(* IEC 61131-3 sources: stc/tests/fixtures/valid_codegen, 3 files *)

(* ---- not_equal.st ---- *)
(* Copyright (C) 2021-2026 Manuele Conti
   SPDX-License-Identifier: GPL-2.0-or-later
   Summary: Verifies code generation for the IEC not-equal operator. *)

FUNCTION differs : BOOL
VAR_INPUT
    left_value, right_value: INT;
END_VAR
    differs := left_value <> right_value;
END_FUNCTION

(* ---- repeat_loop.st ---- *)
(* Copyright (C) 2021-2026 Manuele Conti
   SPDX-License-Identifier: GPL-2.0-or-later
   Summary: Verifies code generation for REPEAT iteration. *)

FUNCTION climb_until : INT
VAR_INPUT
    start_value: INT;
END_VAR
VAR
    cursor_value: INT;
END_VAR
    cursor_value := start_value;
    REPEAT
        cursor_value := cursor_value + 1;
    UNTIL cursor_value >= 10
    END_REPEAT;
    climb_until := cursor_value;
END_FUNCTION

(* ---- typed_literals.st ---- *)
(* Copyright (C) 2021-2026 Manuele Conti
   SPDX-License-Identifier: GPL-2.0-or-later
   Summary: Verifies code generation for typed and based numeric literals. *)

FUNCTION add_literals : INT
VAR_INPUT
    base_value: INT;
END_VAR
    add_literals := base_value + INT#10 + 2#1010 + 16#0A;
END_FUNCTION
